(* CoDeSys 2.3 library: TcSUPS.lib *)
(* Libraries: STANDARD.LIB 5.6.98 11:03:02, TcBase.lib 14.5.09 11:14:08, TcSystem.lib*9.3.10 10:21:30, TcUtilities.lib*8.2.10 16:42:18 *)

(* Global variable list: Global_Variables *)
VAR_GLOBAL
	eGlobalSUpsState	: E_S_UPS_State; (* current ups state of S-UPS *)
END_VAR

(* Data type *)
TYPE E_S_UPS_Mode : (
	eSUPS_WrPersistData_Shutdown,			(* in case of powerfailure: writing of persistent data + shutdown*)
	eSUPS_WrPersistData_NoShutdown,			(* in case of powerfailure: writing of persistent data, no shutdown*)
	eSUPS_ImmediateShutdown,				(* in case of powerfailure: skips writing of data, immediate shutdown*)
	eSUPS_CheckPowerStatus					(* in case of powerfailure: reports powerfailure without action (no writing, no shutdown) *)
);
END_TYPE

(* Data type *)
TYPE E_S_UPS_State : (
	eSUPS_PowerOK,
	eSUPS_PowerFailure,
	eSUPS_WritePersistentData,
	eSUPS_QuickShutdown,
	eSUPS_WaitForRecover,
	eSUPS_WaitForPowerOFF
);


END_TYPE

(* POU F_GetVersionTcSUPS, ST *)
FUNCTION F_GetVersionTcSUPS : UINT	(* Gets the library version info *)
VAR_INPUT
	nVersionElement		:	INT;
(*
	Possible nVersionElement parameter:
	1	:	major number
	2	:	minor number
	3	:	revision number
*)
END_VAR
(* Version history:
Date		|	Version			|	created with					|	Author				|	Remark
dd.mm.yyyy	|					|									|						|
-----------------------------------------------------------------------------------------------------------------------------------------------------------------------------------------------------------------------------------------------------------------------------------
30.11.2009	|	1.0.0			|	TCAT2.11 B1539					|	I.Ch.				|	first release
15.01.2010	|	1.0.1			|	TCAT2.11 B1541					|	I.Ch.				|	global eGlobalSUpsState added
22.03.2010	|	1.0.2			|	TCAT2.11 B1544					|	I.Ch.				|	skip writing/shutdown if powerfail was detected in first scan

*)
CASE nVersionElement OF
1:	(* major number *)
	F_GetVersionTcSUPS := 1;
2:	(* minor number *)
	F_GetVersionTcSUPS := 0;
3:	(* revision number *)
	F_GetVersionTcSUPS := 2;
ELSE
	F_GetVersionTcSUPS := 16#FFFF;
END_CASE
END_FUNCTION

(* POU FB_NT_QuickShutdown, ST *)
FUNCTION_BLOCK FB_NT_QuickShutdown
VAR_INPUT
	NETID				:T_AmsNetId;
	START				:BOOL;
	TMOUT				:TIME := DEFAULT_ADS_TIMEOUT;
END_VAR
VAR_OUTPUT
	BUSY				:BOOL;
	ERR					:BOOL;
	ERRID				:UDINT;
END_VAR
{library private}
VAR
	ADSWRTCTL1			:ADSWRTCTL;
	RisingEdge			:R_TRIG;
	DELAY				:DWORD := 16#FFFFFFFF;
END_VAR
RisingEdge(CLK:=START);

IF RisingEdge.Q THEN
	ADSWRTCTL1(	NETID := NETID,
					PORT := AMSPORT_R3_SYSSERV,
					ADSSTATE := ADSSTATE_POWERFAILURE,
					DEVSTATE := 0,
					LEN := SIZEOF(DELAY),
					SRCADDR :=ADR(DELAY),
					Write := TRUE,
					TMOUT := TMOUT
				);
ELSE
	ADSWRTCTL1( Write:=FALSE);
END_IF


BUSY := ADSWRTCTL1.BUSY;
ERR := ADSWRTCTL1.ERR;
ERRID := ADSWRTCTL1.ERRID;
END_FUNCTION_BLOCK

(* POU FB_S_UPS, ST *)
FUNCTION_BLOCK FB_S_UPS
VAR_INPUT
	sNetID					: T_AmsNetId 		:= ''; 								(* '' = local netid *)
	iPLCPort				: UINT 				:= AMSPORT_R0_PLC_RTS1;				(* PLC Runtime System for writing persistent data *)
	iUPSPort				: UINT 				:= 16#4A8;							(* Port for reading Power State of UPS, dafault 16#4A8 *)
	tTimeout				: TIME 				:= DEFAULT_ADS_TIMEOUT;				(* ADS Timeout *)
	eUpsMode				: E_S_UPS_Mode		:= eSUPS_WrPersistData_Shutdown;	(* UPS mode (w/wo writing persistent data, w/wo shutdown) *)
	ePersistentMode			: E_PersistentMode	:= SPDM_2PASS;						(* mode for writing persistent data *)
	tRecoverTime			: TIME 				:= T#10s;							(* ON time to recover from short power failure in mode eSUPS_WrPersistData_NoShutdown/eSUPS_CheckPowerStatus  *)
END_VAR
VAR_OUTPUT
	bPowerFailDetect		: BOOL;													(* TRUE while powerfailure is detected *)
	eState					: E_S_UPS_State;										(* current ups state *)
END_VAR
{library private}
VAR
	fbWritePersistentData	: FB_WritePersistentData;
	fbNT_QuickShutdown 		: FB_NT_QuickShutdown;
	dwTemp					: DWORD;
	WaitForOffTimer			: TON;
	bFirstCycle				: BOOL := TRUE;
	bPowerOKInFirstCycle	: BOOL := FALSE;
END_VAR
(* monitor power state *)
dwTemp := FW_PortRead(iUPSPort, NoOfByte_DWord);
bPowerFailDetect := dwTemp.0;

(* load check *)
IF bFirstCycle THEN
	bFirstCycle 			:= FALSE;
	bPowerOKInFirstCycle 	:= NOT bPowerFailDetect;
END_IF

(* UPS State Machine *)
CASE eState OF
eSUPS_PowerOK:
	IF bPowerFailDetect THEN
		eState := eSUPS_PowerFailure; 		(* report powerfailure *)
		WaitForOffTimer(IN := FALSE, PT := tRecoverTime);
	END_IF


eSUPS_PowerFailure:
	IF bPowerOKInFirstCycle THEN
		(* allow saving/shutdown because S-UPS is fully loaded *)
		CASE eUpsMode OF
		eSUPS_WrPersistData_Shutdown,			(* in case of powerfailure: writing of persistent data + shutdown *)
		eSUPS_WrPersistData_NoShutdown:			(* in case of powerfailure: writing of persistent data, no shutdown *)
			(* start writing of persistent data *)
			fbWritePersistentData(
				NETID	:= sNetID,
				PORT	:= iPLCPort,
				START	:= TRUE,
				TMOUT	:= tTimeout,
				MODE	:= ePersistentMode
			);
			eState := eSUPS_WritePersistentData;


		eSUPS_CheckPowerStatus:					(* in case of powerfailure: reports powerfailure without action (no writing, no shutdown) *)
			(* check if power recovers *)
			eState := eSUPS_WaitForRecover;


		eSUPS_ImmediateShutdown:				(* in case of powerfailure: skips writing of data, immediate shutdown *)
			(* start quick shutdown *)
			fbNT_QuickShutdown(
				NETID := sNetID,
				START := TRUE,
				TMOUT := tTimeout
			);
			eState := eSUPS_QuickShutdown;

		END_CASE
	ELSE
		(* don't allow saving/shutdown because S-UPS was not fully loaded, just wait for OFF *)
		eState := eSUPS_WaitForPowerOFF;
	END_IF

eSUPS_WritePersistentData:
	(* writing of persistent data *)
	fbWritePersistentData(START	:= FALSE);

	IF eUpsMode = eSUPS_WrPersistData_NoShutdown THEN
		IF NOT fbWritePersistentData.BUSY THEN
			fbWritePersistentData(START	:= FALSE);

			(* wait for OFF *)
			eState := eSUPS_WaitForRecover;
			WaitForOffTimer(IN := FALSE, PT := tRecoverTime);
		END_IF
	ELSE
		IF NOT fbWritePersistentData.BUSY THEN
			fbWritePersistentData(START	:= FALSE);

			(* start quick shutdown *)
			fbNT_QuickShutdown(
				NETID := sNetID,
				START := TRUE,
				TMOUT := tTimeout
			);
			eState := eSUPS_QuickShutdown;
		END_IF
	END_IF


eSUPS_WaitForRecover:
	WaitForOffTimer(IN := (NOT bPowerFailDetect));
	IF WaitForOffTimer.Q THEN
		eState := eSUPS_PowerOK; 		(* report powerOK *)
	END_IF


eSUPS_QuickShutdown:
	(* quick shutdown *)
	fbNT_QuickShutdown(START := FALSE);
	IF NOT fbNT_QuickShutdown.BUSY THEN
		fbNT_QuickShutdown(START := FALSE);

		(* wait for OFF *)
		eState := eSUPS_WaitForPowerOFF;
	END_IF


eSUPS_WaitForPowerOFF:
	(* wait for OFF *)
	eState := eSUPS_WaitForPowerOFF;

END_CASE

eGlobalSUpsState := eState;
END_FUNCTION_BLOCK
